// TIA Portal project "Bachelorarbeit Adrian Gehrig" (V15.1)
// Umsetzung des Smith Prädictor

(* hardware
DEVICE "S71500/ET200MP-Station_1"  S7-1500 station
   slot 0: "Profilschiene_0"  Rack  6ES7 590-1***0-0AA0
   slot 0: "PS 25W 24VDC_1"  PS 25W 24VDC  6ES7 505-0KA00-0AB0  V1.0
   slot 1: "PLC_1"  CPU 1515-2 PN  6ES7 515-2AM01-0AB0  V2.6
      slot 3: "CPU-Display_1"  6ES7591-1BA00-0AA0
*)

// ===== PLC "PLC_1"  CPU 1515-2 PN =====

TYPE "c_c_recursiveEstimat"
// *
//  * File: Smith_Predictor_MIAC.scl
//  *
//  * IEC 61131-3 Structured Text (ST) code generated for subsystem "Smith_Predictor_MIAC/Smith_Predictor_MIAC"
//  *
//  * Model name                      : Smith_Predictor_MIAC
//  * Model version                   : 1.3
//  * Model creator                   : Trips
//  * Model last modified by          : Trips
//  * Model last modified on          : Wed Mar 06 13:07:35 2019
//  * Model sample time               : 0s
//  * Subsystem name                  : Smith_Predictor_MIAC/Smith_Predictor_MIAC
//  * Subsystem sample time           : 1s
//  * Simulink PLC Coder version      : 2.6 (R2018b) 24-May-2018
//  * ST code generated on            : Wed Mar 06 13:15:01 2019
//  *
//  * Target IDE selection            : Siemens SIMATIC Step 7
//  * Test Bench included             : No
//  *
   STRUCT
      IteratorPosition : DInt;
   END_STRUCT;
END_TYPE

TYPE "c_d_recursiveEstimat"
   STRUCT
      OutputDataIterator : "c_c_recursiveEstimat";
      InputDataIterator : "c_c_recursiveEstimat";
   END_STRUCT;
END_TYPE

DATA_BLOCK "PT1_DB"   // DB1
{ S7_Optimized_Access := 'TRUE' }
VERSION : 0.1
// stored: InstanceOfName PT1
"PT1"
BEGIN
END_DATA_BLOCK

DATA_BLOCK "Signale"   // DB2
{ S7_Optimized_Access := 'TRUE' }
VERSION : 0.1
   VAR
      Input_PT1 : Real;
      Input_FOPDT : Real;
      Output_PT1 : Real;
      Output_FOPDT : Real;
      ssMethodType : Int;
      setpoint : Real;
      Start_Adaptation : Real;
      Hand_Value : Real;
      Enable_Auto : Real;
      Start_Identification : Real;
      Gain_Filtered : Real;
      Gain_Not_Filtered : Real;
      pulse_Indicatior : Bool;
      P_Controller : Real;
      I_Controller : Real;
   END_VAR
BEGIN
END_DATA_BLOCK

DATA_BLOCK "FOPDT_DB"   // DB3
{ S7_Optimized_Access := 'TRUE' }
VERSION : 0.1
// stored: InstanceOfName FOPDT
"FOPDT"
BEGIN
END_DATA_BLOCK

DATA_BLOCK "c_Smith_Predictor_MI_DB"   // DB4
{ S7_Optimized_Access := 'TRUE' }
VERSION : 0.1
// stored: InstanceOfName c_Smith_Predictor_MI
"c_Smith_Predictor_MI"
BEGIN
END_DATA_BLOCK

DATA_BLOCK "FOPDT_Tustin0_DB"   // DB5
{ S7_Optimized_Access := 'TRUE' }
VERSION : 0.1
// stored: InstanceOfName FOPDT_Tustin0
"FOPDT_Tustin0"
BEGIN
END_DATA_BLOCK

FUNCTION_BLOCK "PT1"   // FB1, SCL
{ S7_Optimized_Access := 'TRUE' }
VERSION : 0.1
// *
//  * File: TestPLCCoder.scl
//  *
//  * IEC 61131-3 Structured Text (ST) code generated for subsystem "TestPLCCoder/PT1"
//  *
//  * Model name                      : TestPLCCoder
//  * Model version                   : 1.1
//  * Model creator                   : Trips
//  * Model last modified by          : Trips
//  * Model last modified on          : Mon Feb 04 14:14:27 2019
//  * Model sample time               : 0.1s
//  * Subsystem name                  : TestPLCCoder/PT1
//  * Subsystem sample time           : 0.1s
//  * Simulink PLC Coder version      : 2.6 (R2018b) 24-May-2018
//  * ST code generated on            : Wed Feb 06 16:13:48 2019
//  *
//  * Target IDE selection            : Siemens SIMATIC Step 7
//  * Test Bench included             : No
//  *
   VAR_INPUT
      ssMethodType : Int;
      In1 : Real;
   END_VAR
   VAR_OUTPUT
      Out1 : Real;
   END_VAR
   VAR
      c_DiscreteTransferFc : Real;
   END_VAR
BEGIN
   CASE #ssMethodType OF
       0:
           (* InitializeConditions for DiscreteTransferFcn: '<S1>/Discrete Transfer Fcn1' *)
           #c_DiscreteTransferFc := 0.0;
       1:
           (* Outport: '<Root>/Out1' incorporates:
            *  DiscreteTransferFcn: '<S1>/Discrete Transfer Fcn1' *)
           #Out1 := 0.1 * #c_DiscreteTransferFc;
           (* Update for DiscreteTransferFcn: '<S1>/Discrete Transfer Fcn1' *)
           #c_DiscreteTransferFc := #In1 - (-0.9 * #c_DiscreteTransferFc);
   END_CASE;
END_FUNCTION_BLOCK

FUNCTION_BLOCK "FOPDT"   // FB2, SCL
{ S7_Optimized_Access := 'TRUE' }
VERSION : 0.1
// *
//  * File: FOPDT.scl
//  *
//  * IEC 61131-3 Structured Text (ST) code generated for subsystem "FOPDT/Subsystem"
//  *
//  * Model name                      : FOPDT
//  * Model version                   : 1.2
//  * Model creator                   : Trips
//  * Model last modified by          : Trips
//  * Model last modified on          : Tue Feb 26 09:05:07 2019
//  * Model sample time               : 1s
//  * Subsystem name                  : FOPDT/Subsystem
//  * Subsystem sample time           : 1s
//  * Simulink PLC Coder version      : 2.6 (R2018b) 24-May-2018
//  * ST code generated on            : Tue Feb 26 09:08:10 2019
//  *
//  * Target IDE selection            : Siemens SIMATIC Step 7
//  * Test Bench included             : No
//  *
   VAR_INPUT
      ssMethodType : Int;
      FOPD_Input : Real;
      Gain_System1 : Real;
      c_Time_Constant_Syst : Real;
      Sample_Time : Real;
      Dead_Time : DInt;
   END_VAR
   VAR_OUTPUT
      FOPD_Output : Real;
   END_VAR
   VAR
      Divide : Real;
      DiscreteTransferFcnv : Real;
      c_TmpSignalConversio : Array[0..1] of Real;
      Delay_DSTATE : Array[0..799] of Real;
      c_rtb_DiscreteTransf : Real;
      b_i : DInt;
   END_VAR
BEGIN
   CASE #ssMethodType OF
       0:
           (* InitializeConditions for DiscreteTransferFcn: '<S1>/Discrete Transfer Fcn' *)
           #DiscreteTransferFcnv := 0.0;
           (* InitializeConditions for Delay: '<S1>/Delay' *)
           FOR #b_i := 0 TO 799 DO
               #Delay_DSTATE[#b_i] := 0.0;
           END_FOR;
           (* End of InitializeConditions for Delay: '<S1>/Delay' *)
       1:
           (* Product: '<S1>/Divide' *)
           #Divide := #Gain_System1 / #c_Time_Constant_Syst;
           (* SignalConversion: '<S1>/TmpSignal ConversionAtDiscrete Transfer FcnInport3' incorporates:
            *  Constant: '<S1>/Constant'
            *  Gain: '<S1>/Gain'
            *  Gain: '<S1>/Gain1'
            *  Math: '<S1>/Exp'
            *  Product: '<S1>/Divide1'
            *
            * About '<S1>/Exp':
            *  Operator: exp *)
           #c_TmpSignalConversio[0] := 1.0;
           #c_TmpSignalConversio[1] := - EXP((- #Sample_Time) / #c_Time_Constant_Syst);
           (* DiscreteTransferFcn: '<S1>/Discrete Transfer Fcn' *)
           #c_rtb_DiscreteTransf := #Divide * #DiscreteTransferFcnv;
           (* Delay: '<S1>/Delay' *)
           IF #Dead_Time <= 0 THEN
               (* Outport: '<Root>/FOPD_Output' *)
               #FOPD_Output := #c_rtb_DiscreteTransf;
           ELSE
               IF #Dead_Time > 800 THEN
                   #b_i := 800;
               ELSE
                   #b_i := #Dead_Time;
               END_IF;
               (* Outport: '<Root>/FOPD_Output' *)
               #FOPD_Output := #Delay_DSTATE[800 - #b_i];
           END_IF;
           (* End of Delay: '<S1>/Delay' *)

           (* Update for DiscreteTransferFcn: '<S1>/Discrete Transfer Fcn' *)
           #DiscreteTransferFcnv := #FOPD_Input - (#c_TmpSignalConversio[1] * #DiscreteTransferFcnv);
           (* Update for Delay: '<S1>/Delay' *)
           FOR #b_i := 0 TO 798 DO
               #Delay_DSTATE[#b_i] := #Delay_DSTATE[#b_i + 1];
           END_FOR;
           #Delay_DSTATE[799] := #c_rtb_DiscreteTransf;
           (* End of Update for Delay: '<S1>/Delay' *)
   END_CASE;
END_FUNCTION_BLOCK

FUNCTION_BLOCK "ZCFCN_d_RISING"   // FB3, SCL
{ S7_Optimized_Access := 'TRUE' }
VERSION : 0.1
   VAR_INPUT
      u0 : Int;
      u1 : Real;
   END_VAR
   VAR_OUTPUT
      y0 : DInt;
      y1 : Int;
   END_VAR
   VAR
      rising : Bool;
      temp1 : Bool;
      temp2 : Bool;
   END_VAR
BEGIN
   #temp1 := FALSE;
   IF #u1 > 0.0 THEN
       #y1 := 1;
   ELSIF #u1 < 0.0 THEN
       #y1 := 2;
   ELSE
       #y1 := 0;
   END_IF;
   #temp2 := FALSE;
   IF #u0 = 2 THEN
       IF #y1 = 0 THEN
           #rising := TRUE;
       ELSIF #y1 = 1 THEN
           #rising := TRUE;
       ELSE
           #temp2 := TRUE;
       END_IF;
   ELSE
       #temp2 := TRUE;
   END_IF;
   IF #temp2 THEN
       IF #u0 = 0 THEN
           IF #y1 = 1 THEN
               #rising := TRUE;
           ELSE
               #temp1 := TRUE;
           END_IF;
       ELSE
           #temp1 := TRUE;
       END_IF;
   END_IF;
   IF #temp1 THEN
       IF #u0 = 101 THEN
           IF #y1 = 1 THEN
               #rising := TRUE;
           ELSE
               #rising := FALSE;
           END_IF;
       ELSE
           #rising := FALSE;
       END_IF;
   END_IF;
   IF #rising THEN
       #y0 := 1;
   ELSE
       #y0 := 0;
   END_IF;
   IF (#u0 = 2) AND (#y1 = 0) THEN
       #y1 := 100;
   END_IF;
END_FUNCTION_BLOCK

FUNCTION_BLOCK "Smith_Predictor_andv"   // FB4, SCL
{ S7_Optimized_Access := 'TRUE' }
VERSION : 0.1
   VAR_INPUT
      ssMethodType : Int;
      setpoint : Real;
      Dead_Time : Real;
      Y_Process : Real;
      Start_Adaption : Real;
      Hand_Value : Real;
      P_Controller : Real;
      I_Controller : Real;
      Gain_System : Real;
      Time_Constant_System : Real;
      Sample_Time : Real;
      Enable_Auto : Real;
      Start_Identification : Real;
   END_VAR
   VAR_OUTPUT
      Gain_Filtered : Real;
      Gain_Not_Filtered : Real;
      Controller_Output : Real;
   END_VAR
   VAR
      UnitDelay_DSTATE : Real;
      c_Numerator_ZTransfo : Real;
      c_Integrator_IC_LOAD : Int;
      Integrator_DSTATE : Real;
      c_Integrator_PrevRes : Int;
      c_inputSignalLowPass : Real;
      d_outputSignalLowPas : Real;
      icLoad : Int;
      icLoad_o : Int;
      icLoad_g : Int;
      icLoad_m : Int;
      icLoad_k : Int;
      icLoad_f : Int;
      c_EstimatedGainTiefp : Real;
      In1_i : Real;
      In1 : Real;
      In1_m : Real;
      c_System_Simulaton_s : Real;
      In1_b : Real;
      c_arxEstimator_not_e : Bool;
      arxEstimator : "c_d_recursiveEstimat";
      d_inputSignalLowPass : Int := 3;
      e_outputSignalLowPas : Int := 3;
      delayTheta_Reset_ZCE : Int := 3;
      delayL_Reset_ZCE : Int := 3;
      delayPhi_Reset_ZCE : Int := 3;
      c_delayBufferU_Reset : Int := 3;
      c_delayBufferY_Reset : Int := 3;
      c_delayBufferRegress : Int := 3;
      Delay_Reset_ZCE : Int := 3;
      d_EstimatedGainTiefp : Int := 3;
      c_System_Delay_Simul : Int := 3;
      c_System_Simulaton_R : Int := 3;
      d_System_Delay_Simul : Int := 3;
      e_System_Delay_Simul : Array[0..799] of Real;
      f_System_Delay_Simul : Array[0..799] of Real;
      c_Denumerator_ZTrans : Array[0..1] of Real;
      delayL_DSTATE : Array[0..8] of Real;
      delayTheta_DSTATE : Array[0..2] of Real;
      delayPhi_DSTATE : Array[0..3] of Real;
      c_InitialCovariancev : Array[0..8] of Real;
      i0_ZCFCN_d_RISING : "ZCFCN_d_RISING";
      phi : Array[0..2] of Real;
      fTr : Array[0..2] of Real;
      a1 : Real;
      sqrtA0overA1 : Real;
      sqrtA0timesA1 : Real;
      b_kk : DInt;
      rtb_UnitDelay : Real;
      rtb_theta : Array[0..2] of Real;
      rtb_L : Array[0..8] of Real;
      rtb_phiMemory : Array[0..3] of Real;
      imputdelayedminus : Real;
      input : Real;
      c_outputSignalLowPas : Real;
      rtb_theta_tmp : Real;
      rtb_theta_tmp_0 : Real;
   END_VAR
   // c_InitialCovariancev[0] := 3.162278;
   // c_InitialCovariancev[1] := 0.0;
   // c_InitialCovariancev[2] := 0.0;
   // c_InitialCovariancev[3] := 0.0;
   // c_InitialCovariancev[4] := 3.162278;
   // c_InitialCovariancev[5] := 0.0;
   // c_InitialCovariancev[6] := 0.0;
   // c_InitialCovariancev[7] := 0.0;
   // c_InitialCovariancev[8] := 3.162278;
BEGIN
   CASE #ssMethodType OF
       0:
           (* InitializeConditions for UnitDelay: '<S1>/Unit Delay' *)
           #UnitDelay_DSTATE := 0.0;
           (* SystemInitialize for Atomic SubSystem: '<S1>/System Identification' *)
           (* InitializeConditions for DiscreteTransferFcn: '<S3>/input Signal Low Pass Filter' *)
           #c_inputSignalLowPass := 0.0;
           (* InitializeConditions for DiscreteTransferFcn: '<S3>/output Signal Low Pass Filter1' *)
           #d_outputSignalLowPas := 0.0;
           (* InitializeConditions for Delay: '<S106>/delayTheta' *)
           #icLoad := 1;
           (* InitializeConditions for Delay: '<S106>/delayL' *)
           #icLoad_o := 1;
           (* InitializeConditions for Delay: '<S106>/delayPhi' *)
           #icLoad_g := 1;
           (* InitializeConditions for Delay: '<S106>/delayBufferU' *)
           #icLoad_m := 1;
           (* InitializeConditions for Delay: '<S106>/delayBufferY' *)
           #icLoad_k := 1;
           (* InitializeConditions for Delay: '<S126>/delayBufferRegressors' *)
           #icLoad_f := 1;
           (* InitializeConditions for DiscreteTransferFcn: '<S3>/Estimated Gain Tiefpassfilter' *)
           #c_EstimatedGainTiefp := 0.0;
           (* SystemInitialize for MATLAB Function: '<S126>/rarx' *)
           #c_arxEstimator_not_e := FALSE;
           (* SystemInitialize for Enabled SubSystem: '<S3>/Get_Current_Output_Offset' *)
           (* SystemInitialize for Outport: '<S104>/Hold when disabled' *)
           #In1_i := 0.0;
           (* End of SystemInitialize for SubSystem: '<S3>/Get_Current_Output_Offset' *)

           (* SystemInitialize for Enabled SubSystem: '<S3>/Get_Current_delayed_Input_Offset' *)
           (* SystemInitialize for Outport: '<S105>/Hold when disabled' *)
           #In1 := 0.0;
           (* End of SystemInitialize for SubSystem: '<S3>/Get_Current_delayed_Input_Offset' *)
           (* End of SystemInitialize for SubSystem: '<S1>/System Identification' *)

           (* SystemInitialize for Atomic SubSystem: '<S1>/Adaptive SmithPredictor1' *)
           (* InitializeConditions for DiscreteTransferFcn: '<S2>/System_Simulaton' *)
           #c_System_Simulaton_s := 0.0;
           (* End of SystemInitialize for SubSystem: '<S1>/Adaptive SmithPredictor1' *)
           (* SystemInitialize for Atomic SubSystem: '<S1>/Adaptive SmithPredictor1' *)
           (* SystemInitialize for Atomic SubSystem: '<S1>/System Identification' *)
           FOR #b_kk := 0 TO 799 DO
               (* InitializeConditions for Delay: '<S3>/System_Delay_Simulation' *)
               #e_System_Delay_Simul[#b_kk] := 0.0;
               (* InitializeConditions for Delay: '<S2>/System_Delay_Simulation' *)
               #f_System_Delay_Simul[#b_kk] := 0.0;
           END_FOR;
           (* End of SystemInitialize for SubSystem: '<S1>/System Identification' *)

           (* InitializeConditions for DiscreteIntegrator: '<S61>/Integrator' *)
           #c_Integrator_IC_LOAD := 1;
           #c_Integrator_PrevRes := 2;
           (* SystemInitialize for Enabled SubSystem: '<S2>/Get_Current_Offset1' *)
           (* SystemInitialize for Outport: '<S5>/Hold when disabled' *)
           #In1_m := 0.0;
           (* End of SystemInitialize for SubSystem: '<S2>/Get_Current_Offset1' *)

           (* SystemInitialize for Enabled SubSystem: '<S2>/Get_Current_Offset' *)
           (* SystemInitialize for Outport: '<S4>/Hold when disabled' *)
           #In1_b := 0.0;
           (* End of SystemInitialize for SubSystem: '<S2>/Get_Current_Offset' *)
           (* End of SystemInitialize for SubSystem: '<S1>/Adaptive SmithPredictor1' *)
       1:
           (* UnitDelay: '<S1>/Unit Delay' *)
           #rtb_UnitDelay := #UnitDelay_DSTATE;
           (* Outputs for Atomic SubSystem: '<S1>/System Identification' *)
           (* DiscreteTransferFcn: '<S3>/input Signal Low Pass Filter' *)
           #i0_ZCFCN_d_RISING(u0 := #d_inputSignalLowPass,
                              u1 := #Start_Identification);
           #b_kk := #i0_ZCFCN_d_RISING.y0;
           #d_inputSignalLowPass := #i0_ZCFCN_d_RISING.y1;
           IF #b_kk <> 0 THEN
               #c_inputSignalLowPass := 0.0;
           END_IF;
           #input := 0.01 * #c_inputSignalLowPass;
           (* End of DiscreteTransferFcn: '<S3>/input Signal Low Pass Filter' *)

           (* DiscreteTransferFcn: '<S3>/output Signal Low Pass Filter1' *)
           #i0_ZCFCN_d_RISING(u0 := #e_outputSignalLowPas,
                              u1 := #Start_Identification);
           #b_kk := #i0_ZCFCN_d_RISING.y0;
           #e_outputSignalLowPas := #i0_ZCFCN_d_RISING.y1;
           IF #b_kk <> 0 THEN
               #d_outputSignalLowPas := 0.0;
           END_IF;
           #imputdelayedminus := 0.01 * #d_outputSignalLowPas;
           #c_outputSignalLowPas := #imputdelayedminus;
           (* Delay: '<S106>/delayTheta' *)
           #i0_ZCFCN_d_RISING(u0 := #delayTheta_Reset_ZCE,
                              u1 := #Start_Identification);
           #b_kk := #i0_ZCFCN_d_RISING.y0;
           #delayTheta_Reset_ZCE := #i0_ZCFCN_d_RISING.y1;
           IF #b_kk <> 0 THEN
               #icLoad := 1;
           END_IF;
           IF #icLoad <> 0 THEN
               #delayTheta_DSTATE[0] := 2.2204460492503131E-16;
               #delayTheta_DSTATE[1] := 2.2204460492503131E-16;
               #delayTheta_DSTATE[2] := 2.2204460492503131E-16;
           END_IF;
           (* Delay: '<S106>/delayL' incorporates:
            *  Constant: '<S106>/InitialCovariance' *)
           #i0_ZCFCN_d_RISING(u0 := #delayL_Reset_ZCE,
                              u1 := #Start_Identification);
           #b_kk := #i0_ZCFCN_d_RISING.y0;
           #delayL_Reset_ZCE := #i0_ZCFCN_d_RISING.y1;
           IF #b_kk <> 0 THEN
               #icLoad_o := 1;
           END_IF;
           IF #icLoad_o <> 0 THEN
               FOR #b_kk := 0 TO 8 DO
                   #delayL_DSTATE[#b_kk] := #c_InitialCovariancev[#b_kk];
               END_FOR;
           END_IF;
           (* Delay: '<S106>/delayPhi' *)
           #i0_ZCFCN_d_RISING(u0 := #delayPhi_Reset_ZCE,
                              u1 := #Start_Identification);
           #b_kk := #i0_ZCFCN_d_RISING.y0;
           #delayPhi_Reset_ZCE := #i0_ZCFCN_d_RISING.y1;
           IF #b_kk <> 0 THEN
               #icLoad_g := 1;
           END_IF;
           IF #icLoad_g <> 0 THEN
               #delayPhi_DSTATE[0] := 0.0;
               #delayPhi_DSTATE[1] := 0.0;
               #delayPhi_DSTATE[2] := 0.0;
               #delayPhi_DSTATE[3] := 0.0;
           END_IF;
           (* Delay: '<S106>/delayBufferU' *)
           #i0_ZCFCN_d_RISING(u0 := #c_delayBufferU_Reset,
                              u1 := #Start_Identification);
           #b_kk := #i0_ZCFCN_d_RISING.y0;
           #c_delayBufferU_Reset := #i0_ZCFCN_d_RISING.y1;
           IF #b_kk <> 0 THEN
               #icLoad_m := 1;
           END_IF;
           (* End of Delay: '<S106>/delayBufferU' *)

           (* Delay: '<S106>/delayBufferY' *)
           #i0_ZCFCN_d_RISING(u0 := #c_delayBufferY_Reset,
                              u1 := #Start_Identification);
           #b_kk := #i0_ZCFCN_d_RISING.y0;
           #c_delayBufferY_Reset := #i0_ZCFCN_d_RISING.y1;
           IF #b_kk <> 0 THEN
               #icLoad_k := 1;
           END_IF;
           (* End of Delay: '<S106>/delayBufferY' *)

           (* Delay: '<S126>/delayBufferRegressors' *)
           #i0_ZCFCN_d_RISING(u0 := #c_delayBufferRegress,
                              u1 := #Start_Identification);
           #b_kk := #i0_ZCFCN_d_RISING.y0;
           #c_delayBufferRegress := #i0_ZCFCN_d_RISING.y1;
           IF #b_kk <> 0 THEN
               #icLoad_f := 1;
           END_IF;
           (* End of Delay: '<S126>/delayBufferRegressors' *)

           (* Delay: '<S128>/Delay' *)
           #i0_ZCFCN_d_RISING(u0 := #Delay_Reset_ZCE,
                              u1 := #Start_Identification);
           #b_kk := #i0_ZCFCN_d_RISING.y0;
           #Delay_Reset_ZCE := #i0_ZCFCN_d_RISING.y1;
           (* MATLAB Function: '<S126>/rarx' *)
           (* % Was a reset trigered? *)
           (* MATLAB Function 'Recursive Estimation/rarx/rarx': '<S135>:1' *)
           (* Copyright 2015-2018 The MathWorks, Inc. *)
           (* Get the estimator object. Use the arx estimator with nb=0 *)
           (* '<S135>:1:17' if isempty(arxEstimator) *)
           IF NOT #c_arxEstimator_not_e THEN
               (* '<S135>:1:18' arxEstimator = recursiveEstimation.internal.rpoly.getEstimator(... *)
               (* '<S135>:1:19'         'arx',... *)
               (* '<S135>:1:20'         algorithmParams); *)
               #c_arxEstimator_not_e := TRUE;
           END_IF;
           (* If user triggered a reset, communicate this to the estimator *)
           (* '<S135>:1:24' if hasTriggeredReset *)
           (* Update algorithm states, perform estimation *)
           (* % States *)
           (* % new IO data *)
           (* '<S135>:1:31' [phiMemory, uMemory, yMemory, regressorsMemory, ... *)
           (* '<S135>:1:32'     theta, L, ... *)
           (* '<S135>:1:33'     A, B, e] = ... *)
           (* '<S135>:1:34'     arxEstimator.estimate(... *)
           (* '<S135>:1:35'     phiMemory, uMemory, yMemory, regressorsMemory, theta, L, ... % States *)
           (* '<S135>:1:36'     yMeas, uMeas,... % new IO data *)
           (* '<S135>:1:37'     isEnabled, adg1, adg2, algorithmParams); *)
           #arxEstimator.OutputDataIterator.IteratorPosition := 1;
           #arxEstimator.InputDataIterator.IteratorPosition := 1;
           #arxEstimator.OutputDataIterator.IteratorPosition := MIN(IN1 := #arxEstimator.OutputDataIterator.IteratorPosition + 1,
                                                                    IN2 := 2);
           #arxEstimator.InputDataIterator.IteratorPosition := MIN(IN1 := #arxEstimator.InputDataIterator.IteratorPosition + 1,
                                                                   IN2 := 2);
           (* End of Outputs for SubSystem: '<S1>/System Identification' *)
           (* Outputs for Atomic SubSystem: '<S1>/System Identification' *)
           (* MATLAB Function: '<S126>/rarx' incorporates:
            *  DataTypeConversion: '<S106>/DataTypeConversionEnable'
            *  Delay: '<S106>/delayL'
            *  Delay: '<S106>/delayPhi'
            *  Delay: '<S106>/delayTheta'
            *  DiscreteTransferFcn: '<S3>/output Signal Low Pass Filter1' *)
           FOR #b_kk := 0 TO 8 DO
               #rtb_L[#b_kk] := #delayL_DSTATE[#b_kk];
           END_FOR;
           #rtb_theta[0] := #delayTheta_DSTATE[0];
           #rtb_theta[1] := #delayTheta_DSTATE[1];
           #rtb_theta[2] := #delayTheta_DSTATE[2];
           #imputdelayedminus := #imputdelayedminus - (((#delayPhi_DSTATE[0] * #delayTheta_DSTATE[0]) + (#delayPhi_DSTATE[1] * #delayTheta_DSTATE[1])
           ) + (#delayPhi_DSTATE[3] * #delayTheta_DSTATE[2]));
           IF #Start_Identification <> 0.0 THEN
               FOR #b_kk := 0 TO 2 DO
                   #fTr[#b_kk] := (#delayL_DSTATE[(3 * #b_kk) + 2] * #delayPhi_DSTATE[3]) + ((#delayL_DSTATE[(3 * #b_kk) + 1] * #delayPhi_DSTATE[1])
                   + (#delayL_DSTATE[3 * #b_kk] * #delayPhi_DSTATE[0]));
               END_FOR;
               #phi[0] := 0.0;
               #rtb_theta[0] := 0.0;
               #phi[1] := 0.0;
               #rtb_theta[1] := 0.0;
               #a1 := (#fTr[2] * #fTr[2]) + 1.0;
               #sqrtA0overA1 := SQRT(1.0 / #a1);
               #rtb_theta[2] := #rtb_L[8] * #fTr[2];
               #rtb_L[8] := (#rtb_L[8] * #sqrtA0overA1) - (0.0 / (#sqrtA0overA1 * #a1));
               #phi[2] := #rtb_theta[2];
               #sqrtA0overA1 := #a1;
               #a1 := (#fTr[1] * #fTr[1]) + #a1;
               #sqrtA0overA1 := SQRT(#sqrtA0overA1 / #a1);
               #sqrtA0timesA1 := #sqrtA0overA1 * #a1;
               FOR #b_kk := 0 TO 1 DO
                   #rtb_theta_tmp := #rtb_L[5 - #b_kk];
                   #rtb_theta_tmp_0 := #phi[2 - #b_kk];
                   #rtb_theta[2 - #b_kk] := (#rtb_theta_tmp * #fTr[1]) + #rtb_theta_tmp_0;
                   #rtb_L[5 - #b_kk] := (#rtb_theta_tmp * #sqrtA0overA1) - ((#rtb_theta_tmp_0 * #fTr[1]) / #sqrtA0timesA1);
                   #phi[2 - #b_kk] := #rtb_theta[2 - #b_kk];
               END_FOR;
               #sqrtA0overA1 := #a1;
               #a1 := (#fTr[0] * #fTr[0]) + #a1;
               #sqrtA0overA1 := SQRT(#sqrtA0overA1 / #a1);
               #sqrtA0timesA1 := #sqrtA0overA1 * #a1;
               FOR #b_kk := 0 TO 2 DO
                   #rtb_theta_tmp := #rtb_L[2 - #b_kk];
                   #rtb_theta_tmp_0 := #phi[2 - #b_kk];
                   #rtb_theta[2 - #b_kk] := (#rtb_theta_tmp * #fTr[0]) + #rtb_theta_tmp_0;
                   #rtb_L[2 - #b_kk] := (#rtb_theta_tmp * #sqrtA0overA1) - ((#rtb_theta_tmp_0 * #fTr[0]) / #sqrtA0timesA1);
                   #phi[2 - #b_kk] := #rtb_theta[2 - #b_kk];
               END_FOR;
               #rtb_theta[0] := #rtb_theta[0] / #a1;
               #rtb_theta[1] := #rtb_theta[1] / #a1;
               #rtb_theta[0] := (#rtb_theta[0] * #imputdelayedminus) + #delayTheta_DSTATE[0];
               #rtb_theta[1] := (#rtb_theta[1] * #imputdelayedminus) + #delayTheta_DSTATE[1];
               #rtb_theta[2] := ((#rtb_theta[2] / #a1) * #imputdelayedminus) + #delayTheta_DSTATE[2];
           END_IF;
           #rtb_phiMemory[2] := #delayPhi_DSTATE[1];
           #rtb_phiMemory[1] := #delayPhi_DSTATE[0];
           (* Outputs for Atomic SubSystem: '<S3>/Calculate DC Gain1' *)
           (* Product: '<S103>/Divide' incorporates:
            *  MATLAB Function: '<S126>/rarx'
            *  Sum: '<S103>/A(z) Sum of Elements' *)
            (* helper variables *)
           #a1 := #rtb_theta[2] / ((1.0 + #rtb_theta[0]) + #rtb_theta[1]);
           (* Saturate: '<S103>/Gain_Saturation' incorporates:
            *  Outport: '<Root>/Gain_Filtered' *)
           IF #a1 >= 1.5 THEN
               #Gain_Filtered := 1.5;
           ELSIF #a1 > 0.01 THEN
               #Gain_Filtered := #a1;
           ELSE
               #Gain_Filtered := 0.01;
           END_IF;
           (* End of Saturate: '<S103>/Gain_Saturation' *)
           (* End of Outputs for SubSystem: '<S3>/Calculate DC Gain1' *)

           (* DiscreteTransferFcn: '<S3>/Estimated Gain Tiefpassfilter' incorporates:
            *  Constant: '<S3>/Constant3' *)
           #i0_ZCFCN_d_RISING(u0 := #d_EstimatedGainTiefp,
                              u1 := #Start_Identification);
           #b_kk := #i0_ZCFCN_d_RISING.y0;
           #d_EstimatedGainTiefp := #i0_ZCFCN_d_RISING.y1;
           IF #b_kk <> 0 THEN
               #c_EstimatedGainTiefp := 0.0;
           END_IF;
           #sqrtA0overA1 := 0.00083333333333333339 * #c_EstimatedGainTiefp;
           (* End of DiscreteTransferFcn: '<S3>/Estimated Gain Tiefpassfilter' *)

           (* Outputs for Enabled SubSystem: '<S3>/Get_Current_Output_Offset' incorporates:
            *  EnablePort: '<S104>/Enable' *)
            (* Logic: '<S3>/NOT' incorporates:
             *  Inport: '<S104>/In1' *)
           IF #Start_Identification = 0.0 THEN
               #In1_i := #Y_Process;
           END_IF;
           (* End of Logic: '<S3>/NOT' *)
           (* End of Outputs for SubSystem: '<S3>/Get_Current_Output_Offset' *)

           (* Delay: '<S3>/System_Delay_Simulation' incorporates:
            *  Constant: '<S3>/Vorsicht wenn resettet wird muss erst dieser Totzeitspeicher  voll gelaufen sein bevor die Adaption starten darf  Sonst kommt heir immer 0 raus und die Identifikation kann nicht rechnen' *)
           #i0_ZCFCN_d_RISING(u0 := #c_System_Delay_Simul,
                              u1 := 0.0);
           #b_kk := #i0_ZCFCN_d_RISING.y0;
           #c_System_Delay_Simul := #i0_ZCFCN_d_RISING.y1;
           IF #b_kk <> 0 THEN
               FOR #b_kk := 0 TO 799 DO
                   #e_System_Delay_Simul[#b_kk] := 0.0;
               END_FOR;
           END_IF;
           IF #Dead_Time < 1.0 THEN
               #a1 := #rtb_UnitDelay;
           ELSE
               IF #Dead_Time > 800.0 THEN
                   #b_kk := 800;
               ELSE
                   #b_kk := TRUNC(#Dead_Time);
               END_IF;
               #a1 := #e_System_Delay_Simul[800 - #b_kk];
           END_IF;
           (* End of Delay: '<S3>/System_Delay_Simulation' *)

           (* Outputs for Enabled SubSystem: '<S3>/Get_Current_delayed_Input_Offset' incorporates:
            *  EnablePort: '<S105>/Enable' *)
            (* Logic: '<S3>/NOT1' incorporates:
             *  Inport: '<S105>/In1' *)
           IF #Start_Identification = 0.0 THEN
               #In1 := #a1;
           END_IF;
           (* End of Logic: '<S3>/NOT1' *)
           (* End of Outputs for SubSystem: '<S3>/Get_Current_delayed_Input_Offset' *)

           (* Update for DiscreteTransferFcn: '<S3>/input Signal Low Pass Filter' incorporates:
            *  Sum: '<S3>/Substract Current Offset  so that the linearised model works1' *)
           #c_inputSignalLowPass := (#a1 - #In1) - (-0.99 * #c_inputSignalLowPass);
           (* Update for DiscreteTransferFcn: '<S3>/output Signal Low Pass Filter1' incorporates:
            *  Sum: '<S3>/Substract Current Offset  so that the linearised model works' *)
           #d_outputSignalLowPas := (#Y_Process - #In1_i) - (-0.99 * #d_outputSignalLowPas);
           (* Update for Delay: '<S106>/delayTheta' *)
           #icLoad := 0;
           #delayTheta_DSTATE[0] := #rtb_theta[0];
           #delayTheta_DSTATE[1] := #rtb_theta[1];
           #delayTheta_DSTATE[2] := #rtb_theta[2];
           (* Update for Delay: '<S106>/delayL' *)
           #icLoad_o := 0;
           (* End of Outputs for SubSystem: '<S1>/System Identification' *)
           (* Outputs for Atomic SubSystem: '<S1>/System Identification' *)
           (* Update for Delay: '<S106>/delayL' *)
           FOR #b_kk := 0 TO 8 DO
               #delayL_DSTATE[#b_kk] := #rtb_L[#b_kk];
           END_FOR;
           (* Update for Delay: '<S106>/delayPhi' incorporates:
            *  MATLAB Function: '<S126>/rarx' *)
           #icLoad_g := 0;
           #delayPhi_DSTATE[0] := - #c_outputSignalLowPas;
           #delayPhi_DSTATE[1] := #rtb_phiMemory[1];
           #delayPhi_DSTATE[2] := #rtb_phiMemory[2];
           #delayPhi_DSTATE[3] := #input;
           (* Update for Delay: '<S106>/delayBufferU' *)
           #icLoad_m := 0;
           (* Update for Delay: '<S106>/delayBufferY' *)
           #icLoad_k := 0;
           (* Update for Delay: '<S126>/delayBufferRegressors' *)
           #icLoad_f := 0;
           (* Update for DiscreteTransferFcn: '<S3>/Estimated Gain Tiefpassfilter' incorporates:
            *  Outport: '<Root>/Gain_Filtered' *)
           #c_EstimatedGainTiefp := #Gain_Filtered - (-0.99916701379245831 * #c_EstimatedGainTiefp);
           (* Update for Delay: '<S3>/System_Delay_Simulation' *)
           FOR #b_kk := 0 TO 798 DO
               #e_System_Delay_Simul[#b_kk] := #e_System_Delay_Simul[#b_kk + 1];
           END_FOR;
           #e_System_Delay_Simul[799] := #rtb_UnitDelay;
           (* End of Update for Delay: '<S3>/System_Delay_Simulation' *)
           (* End of Outputs for SubSystem: '<S1>/System Identification' *)

           (* Outport: '<Root>/Gain_Not_Filtered' *)
           #Gain_Not_Filtered := #sqrtA0overA1;
           (* Outputs for Atomic SubSystem: '<S1>/Adaptive SmithPredictor1' *)
           (* Product: '<S2>/Divide' incorporates:
            *  Constant: '<S2>/Constant1' *)
           #c_Numerator_ZTransfo := 1.0 / #Time_Constant_System;
           (* Switch: '<S2>/Hand_Mode2' incorporates:
            *  Constant: '<S2>/Constant2' *)
           IF #Enable_Auto > 0.0 THEN
               #a1 := #setpoint;
           ELSE
               #a1 := 0.0;
           END_IF;
           (* End of Switch: '<S2>/Hand_Mode2' *)

           (* Outputs for Enabled SubSystem: '<S2>/Get_Current_Offset1' incorporates:
            *  EnablePort: '<S5>/Enable' *)
            (* Logic: '<S2>/NOT1' incorporates:
             *  Inport: '<S5>/In1' *)
           IF #Enable_Auto = 0.0 THEN
               #In1_m := #Y_Process;
           END_IF;
           (* End of Logic: '<S2>/NOT1' *)
           (* End of Outputs for SubSystem: '<S2>/Get_Current_Offset1' *)

           (* Switch: '<S2>/Hand_Mode4' incorporates:
            *  Constant: '<S2>/Constant5' *)
           IF #Enable_Auto > 0.0 THEN
               #rtb_UnitDelay := #In1_m;
           ELSE
               #rtb_UnitDelay := 0.0;
           END_IF;
           (* End of Switch: '<S2>/Hand_Mode4' *)

           (* Sum: '<S2>/Substract Current Setpoint Offset' *)
           #c_outputSignalLowPas := #a1 - #rtb_UnitDelay;
           (* SignalConversion: '<S2>/TmpSignal ConversionAtSystem_SimulatonInport3' incorporates:
            *  Constant: '<S2>/Constant'
            *  Gain: '<S2>/Gain'
            *  Gain: '<S2>/Gain1'
            *  Math: '<S2>/Exp'
            *  Product: '<S2>/Divide1'
            *
            * About '<S2>/Exp':
            *  Operator: exp *)
           #c_Denumerator_ZTrans[0] := 1.0;
           #c_Denumerator_ZTrans[1] := - EXP((- #Sample_Time) / #Time_Constant_System);
           (* DiscreteTransferFcn: '<S2>/System_Simulaton' *)
           #i0_ZCFCN_d_RISING(u0 := #c_System_Simulaton_R,
                              u1 := #Enable_Auto);
           #b_kk := #i0_ZCFCN_d_RISING.y0;
           #c_System_Simulaton_R := #i0_ZCFCN_d_RISING.y1;
           IF #b_kk <> 0 THEN
               #c_System_Simulaton_s := 0.0;
           END_IF;
           #input := #c_Numerator_ZTransfo * #c_System_Simulaton_s;
           (* End of DiscreteTransferFcn: '<S2>/System_Simulaton' *)

           (* Delay: '<S2>/System_Delay_Simulation' *)
           #i0_ZCFCN_d_RISING(u0 := #d_System_Delay_Simul,
                              u1 := #Enable_Auto);
           #b_kk := #i0_ZCFCN_d_RISING.y0;
           #d_System_Delay_Simul := #i0_ZCFCN_d_RISING.y1;
           IF #b_kk <> 0 THEN
               FOR #b_kk := 0 TO 799 DO
                   #f_System_Delay_Simul[#b_kk] := 0.0;
               END_FOR;
           END_IF;
           IF #Dead_Time < 1.0 THEN
               #imputdelayedminus := #input;
           ELSE
               IF #Dead_Time > 800.0 THEN
                   #b_kk := 800;
               ELSE
                   #b_kk := TRUNC(#Dead_Time);
               END_IF;
               #imputdelayedminus := #f_System_Delay_Simul[800 - #b_kk];
           END_IF;
           (* End of Delay: '<S2>/System_Delay_Simulation' *)

           (* Switch: '<S2>/Hand_Mode3' incorporates:
            *  Constant: '<S2>/Constant3' *)
           IF #Enable_Auto > 0.0 THEN
               #a1 := #Y_Process;
           ELSE
               #a1 := 0.0;
           END_IF;
           (* End of Switch: '<S2>/Hand_Mode3' *)

           (* Sum: '<S2>/Sum' incorporates:
            *  Sum: '<S2>/Substract Current Offset  so that the linearised model works1'
            *  Sum: '<S2>/Sum17'
            *  Sum: '<S2>/Sum18' *)
           #rtb_UnitDelay := #c_outputSignalLowPas - (((#a1 - #rtb_UnitDelay) - #imputdelayedminus) + #input);
           (* DiscreteIntegrator: '<S61>/Integrator' *)
           IF #c_Integrator_IC_LOAD <> 0 THEN
               #Integrator_DSTATE := #Hand_Value;
           END_IF;
           IF (#Enable_Auto > 0.0) AND (#c_Integrator_PrevRes <= 0) THEN
               #Integrator_DSTATE := #Hand_Value;
           END_IF;
           (* Sum: '<S90>/Sum' incorporates:
            *  DiscreteIntegrator: '<S61>/Integrator'
            *  Product: '<S77>/PProd Out' *)
           #a1 := (#rtb_UnitDelay * #P_Controller) + #Integrator_DSTATE;
           (* Saturate: '<S82>/Saturation' *)
           IF #a1 >= 100.0 THEN
               #a1 := 100.0;
           ELSIF #a1 <= 0.0 THEN
               #a1 := 0.0;
           END_IF;
           (* End of Saturate: '<S82>/Saturation' *)

           (* Switch: '<S2>/Hand_Mode' *)
           IF #Enable_Auto > 0.0 THEN
               #Controller_Output := #a1;
           ELSE
               #Controller_Output := #Hand_Value;
           END_IF;
           (* End of Switch: '<S2>/Hand_Mode' *)

           (* Outputs for Enabled SubSystem: '<S2>/Get_Current_Offset' incorporates:
            *  EnablePort: '<S4>/Enable' *)
            (* Logic: '<S2>/NOT' incorporates:
             *  Inport: '<S4>/In1' *)
           IF #Enable_Auto = 0.0 THEN
               #In1_b := #Controller_Output;
           END_IF;
           (* End of Logic: '<S2>/NOT' *)
           (* End of Outputs for SubSystem: '<S2>/Get_Current_Offset' *)

           (* Switch: '<S2>/Hand_Mode1' incorporates:
            *  Constant: '<S2>/Constant4'
            *  Sum: '<S2>/Substract Current Offset  so that the linearised model works' *)
           IF #Enable_Auto > 0.0 THEN
               #a1 := #Controller_Output - #In1_b;
           ELSE
               #a1 := 0.0;
           END_IF;
           (* End of Switch: '<S2>/Hand_Mode1' *)

           (* Switch: '<S2>/Switch_from_initial_Gain_to_Estimated' *)
           IF #Start_Adaption <= 0.0 THEN
               #sqrtA0overA1 := #Gain_System;
           END_IF;
           (* End of Switch: '<S2>/Switch_from_initial_Gain_to_Estimated' *)

           (* Product: '<S2>/Mul_Gain_or_Estimate' *)
           #sqrtA0overA1 := #a1 * #sqrtA0overA1;
           (* Update for DiscreteTransferFcn: '<S2>/System_Simulaton' *)
           #c_System_Simulaton_s := #sqrtA0overA1 - (#c_Denumerator_ZTrans[1] * #c_System_Simulaton_s);
           (* Update for Delay: '<S2>/System_Delay_Simulation' *)
           FOR #b_kk := 0 TO 798 DO
               #f_System_Delay_Simul[#b_kk] := #f_System_Delay_Simul[#b_kk + 1];
           END_FOR;
           #f_System_Delay_Simul[799] := #input;
           (* End of Update for Delay: '<S2>/System_Delay_Simulation' *)

           (* Update for DiscreteIntegrator: '<S61>/Integrator' incorporates:
            *  Product: '<S50>/IProd Out' *)
           #c_Integrator_IC_LOAD := 0;
           #Integrator_DSTATE := (#rtb_UnitDelay * #I_Controller) + #Integrator_DSTATE;
           IF #Enable_Auto > 0.0 THEN
               #c_Integrator_PrevRes := 1;
           ELSIF #Enable_Auto < 0.0 THEN
               #c_Integrator_PrevRes := -1;
           ELSIF #Enable_Auto = 0.0 THEN
               #c_Integrator_PrevRes := 0;
           ELSE
               #c_Integrator_PrevRes := 2;
           END_IF;
           (* End of Update for DiscreteIntegrator: '<S61>/Integrator' *)
           (* End of Outputs for SubSystem: '<S1>/Adaptive SmithPredictor1' *)

           (* Update for UnitDelay: '<S1>/Unit Delay' *)
           #UnitDelay_DSTATE := #Controller_Output;
   END_CASE;
END_FUNCTION_BLOCK

FUNCTION_BLOCK "FOPDT_Tustin0"   // FB5, SCL
{ S7_Optimized_Access := 'TRUE' }
VERSION : 0.1
// *
//  * File: FOPDT_Tustin.scl
//  *
//  * IEC 61131-3 Structured Text (ST) code generated for subsystem "FOPDT_Tustin/FOPDT_Tustin"
//  *
//  * Model name                      : FOPDT_Tustin
//  * Model version                   : 1.11
//  * Model creator                   : Trips
//  * Model last modified by          : Trips
//  * Model last modified on          : Mon Mar 04 23:33:50 2019
//  * Model sample time               : 1s
//  * Subsystem name                  : FOPDT_Tustin/FOPDT_Tustin
//  * Subsystem sample time           : 1s
//  * Simulink PLC Coder version      : 2.6 (R2018b) 24-May-2018
//  * ST code generated on            : Mon Mar 04 23:34:12 2019
//  *
//  * Target IDE selection            : Siemens SIMATIC Step 7
//  * Test Bench included             : No
//  *
   VAR_INPUT
      ssMethodType : Int;
      FOPD_Input : Real;
      Gain_System : Real;
      Time_Constant_System : Real;
      Sample_Time : Real;
      Dead_Time : Real;
   END_VAR
   VAR_OUTPUT
      FOPD_Output : Real;
   END_VAR
   VAR
      DiscreteTransferFcnv : Real;
      c_TmpSignalConversio : Array[0..1] of Real;
      Delay_DSTATE : Array[0..799] of Real;
      d_TmpSignalConversio : Array[0..1] of Real;
      rtb_Gain : Real;
      rtb_Divide : Real;
      b_i : DInt;
   END_VAR
BEGIN
   CASE #ssMethodType OF
       0:
           (* InitializeConditions for DiscreteTransferFcn: '<S1>/Discrete Transfer Fcn' *)
           #DiscreteTransferFcnv := 0.0;
           (* InitializeConditions for Delay: '<S1>/Delay' *)
           FOR #b_i := 0 TO 799 DO
               #Delay_DSTATE[#b_i] := 0.0;
           END_FOR;
           (* End of InitializeConditions for Delay: '<S1>/Delay' *)
       1:
           (* Gain: '<S1>/Gain' *)
           #rtb_Gain := 2.0 * #Time_Constant_System;
           (* Product: '<S1>/Divide' incorporates:
            *  Product: '<S1>/Multiply'
            *  Sum: '<S1>/Add' *)
           #rtb_Divide := (#Gain_System * #Sample_Time) / (#Sample_Time + #rtb_Gain);
           (* SignalConversion: '<S1>/TmpSignal ConversionAtDiscrete Transfer FcnInport2' *)
           #c_TmpSignalConversio[0] := #rtb_Divide;
           #c_TmpSignalConversio[1] := #rtb_Divide;
           (* SignalConversion: '<S1>/TmpSignal ConversionAtDiscrete Transfer FcnInport3' incorporates:
            *  Constant: '<S1>/Constant'
            *  Gain: '<S1>/Gain1'
            *  Product: '<S1>/Divide1'
            *  Sum: '<S1>/Add1'
            *  Sum: '<S1>/Minus' *)
           #d_TmpSignalConversio[0] := 1.0;
           #d_TmpSignalConversio[1] := - ((#rtb_Gain - #Sample_Time) / (#rtb_Gain + #Sample_Time));
           (* DiscreteTransferFcn: '<S1>/Discrete Transfer Fcn' *)
           #rtb_Gain := #FOPD_Input - (#d_TmpSignalConversio[1] * #DiscreteTransferFcnv);
           #rtb_Divide := (#c_TmpSignalConversio[0] * #rtb_Gain) + (#c_TmpSignalConversio[1] * #DiscreteTransferFcnv);
           (* Delay: '<S1>/Delay' *)
           IF #Dead_Time < 1.0 THEN
               (* Outport: '<Root>/FOPD_Output' *)
               #FOPD_Output := #rtb_Divide;
           ELSE
               IF #Dead_Time > 800.0 THEN
                   #b_i := 800;
               ELSE
                   #b_i := TRUNC(#Dead_Time);
               END_IF;
               (* Outport: '<Root>/FOPD_Output' *)
               #FOPD_Output := #Delay_DSTATE[800 - #b_i];
           END_IF;
           (* End of Delay: '<S1>/Delay' *)

           (* Update for DiscreteTransferFcn: '<S1>/Discrete Transfer Fcn' *)
           #DiscreteTransferFcnv := #rtb_Gain;
           (* Update for Delay: '<S1>/Delay' *)
           FOR #b_i := 0 TO 798 DO
               #Delay_DSTATE[#b_i] := #Delay_DSTATE[#b_i + 1];
           END_FOR;
           #Delay_DSTATE[799] := #rtb_Divide;
           (* End of Update for Delay: '<S1>/Delay' *)
   END_CASE;
END_FUNCTION_BLOCK

FUNCTION_BLOCK "c_Smith_Predictor_MI"   // FB6, SCL
{ S7_Optimized_Access := 'TRUE' }
VERSION : 0.1
   VAR_INPUT
      ssMethodType : Int;
      Setpoint : Real;
      Process_Value : Real;
      Gain_System : Real;
      Time_Constant_System : Real;
      Dead_Time_System : DInt;
      Enable_Auto : Real;
      Hand_Value : Real;
      P_Controller : Real;
      I_Controller : Real;
      Start_Identification : Real;
      c_Time_Constant_Gain : Real;
      c_Time_Constant_Esti : Real;
      Enable_Adaption : Real;
      Sample_Time : Real;
   END_VAR
   VAR_OUTPUT
      Gain_NOT_Filtered : Real;
      Gain_Filtered : Real;
      Controller_Value : Real;
   END_VAR
   VAR
      UnitDelay_DSTATE : Real;
      c_Integrator_IC_LOAD : Int;
      Integrator_DSTATE : Real;
      c_Integrator_PrevRes : Int;
      In1 : Real;
      In1_b : Real;
      icLoad : Int;
      icLoad_i : Int;
      icLoad_p : Int;
      icLoad_b : Int;
      icLoad_ih : Int;
      icLoad_n : Int;
      Multiply : Real;
      In1_a : Real;
      In1_n : Real;
      UnitDelay_DSTATE_j : Real;
      c_arxEstimator_not_e : Bool;
      arxEstimator : "c_d_recursiveEstimat";
      DiscreteTransferFcnv : Real;
      b_DiscreteTransferFc : Real;
      c_System_Delay_Simul : Int := 3;
      delayTheta_Reset_ZCE : Int := 3;
      delayL_Reset_ZCE : Int := 3;
      delayPhi_Reset_ZCE : Int := 3;
      c_delayBufferU_Reset : Int := 3;
      c_delayBufferY_Reset : Int := 3;
      c_delayBufferRegress : Int := 3;
      Delay_Reset_ZCE : Int := 3;
      d_System_Delay_Simul : Int := 3;
      c_DiscreteTransferFc : Int := 3;
      d_DiscreteTransferFc : Int := 3;
      e_System_Delay_Simul : Array[0..799] of Real;
      f_System_Delay_Simul : Array[0..799] of Real;
      c_TmpSignalConversio : Array[0..1] of Real;
      d_TmpSignalConversio : Array[0..1] of Real;
      e_TmpSignalConversio : Array[0..1] of Real;
      f_TmpSignalConversio : Array[0..1] of Real;
      delayL_DSTATE : Array[0..8] of Real;
      delayTheta_DSTATE : Array[0..2] of Real;
      delayPhi_DSTATE : Array[0..3] of Real;
      c_InitialCovariancev : Array[0..8] of Real;
      i0_ZCFCN_d_RISING : "ZCFCN_d_RISING";
      i0_PT1_Tustin1 : "PT1_Tustin1";
      i1_PT1_Tustin1 : "PT1_Tustin1";
      phi : Array[0..2] of Real;
      fTr : Array[0..2] of Real;
      a1 : Real;
      sqrtA0overA1 : Real;
      sqrtA0timesA1 : Real;
      b_kk : DInt;
      rtb_UnitDelay : Real;
      rtb_theta : Array[0..2] of Real;
      rtb_AzSumofElements : Real;
      c_rtb_DiscreteTransf : Real;
      d_rtb_DiscreteTransf : Real;
      rtb_L : Array[0..8] of Real;
      rtb_phiMemory : Array[0..3] of Real;
      rtb_theta_tmp : Real;
   END_VAR
   // c_InitialCovariancev[0] := 3.162278;
   // c_InitialCovariancev[1] := 0.0;
   // c_InitialCovariancev[2] := 0.0;
   // c_InitialCovariancev[3] := 0.0;
   // c_InitialCovariancev[4] := 3.162278;
   // c_InitialCovariancev[5] := 0.0;
   // c_InitialCovariancev[6] := 0.0;
   // c_InitialCovariancev[7] := 0.0;
   // c_InitialCovariancev[8] := 3.162278;
BEGIN
   CASE #ssMethodType OF
       0:
           (* InitializeConditions for UnitDelay: '<S1>/Unit Delay' *)
           #UnitDelay_DSTATE := 0.0;
           (* SystemInitialize for Atomic SubSystem: '<S1>/System Identification' *)
           (* InitializeConditions for Delay: '<S3>/System_Delay_Simulation' *)
           FOR #b_kk := 0 TO 799 DO
               #e_System_Delay_Simul[#b_kk] := 0.0;
           END_FOR;
           (* End of InitializeConditions for Delay: '<S3>/System_Delay_Simulation' *)

           (* InitializeConditions for Delay: '<S110>/delayTheta' *)
           #icLoad := 1;
           (* InitializeConditions for Delay: '<S110>/delayL' *)
           #icLoad_i := 1;
           (* InitializeConditions for Delay: '<S110>/delayPhi' *)
           #icLoad_p := 1;
           (* InitializeConditions for Delay: '<S110>/delayBufferU' *)
           #icLoad_b := 1;
           (* InitializeConditions for Delay: '<S110>/delayBufferY' *)
           #icLoad_ih := 1;
           (* InitializeConditions for Delay: '<S130>/delayBufferRegressors' *)
           #icLoad_n := 1;
           (* SystemInitialize for Enabled SubSystem: '<S3>/Get_Current_delayed_Input_Offset' *)
           (* SystemInitialize for Outport: '<S106>/Hold when disabled' *)
           #In1 := 0.0;
           (* End of SystemInitialize for SubSystem: '<S3>/Get_Current_delayed_Input_Offset' *)
           (* End of SystemInitialize for SubSystem: '<S1>/System Identification' *)

           (* Constant: '<S3>/Constant2' *)
           #i0_PT1_Tustin1(ssMethodType := 0,
                           PT1_Input := #a1,
                           Gain_System := 1.0,
                           Time_Constant_System := #c_Time_Constant_Esti,
                           Reset := #Start_Identification);
           (* SystemInitialize for Atomic SubSystem: '<S1>/System Identification' *)
           (* SystemInitialize for Enabled SubSystem: '<S3>/Get_Current_Output_Offset' *)
           (* SystemInitialize for Outport: '<S105>/Hold when disabled' *)
           #In1_b := 0.0;
           (* End of SystemInitialize for SubSystem: '<S3>/Get_Current_Output_Offset' *)
           (* End of SystemInitialize for SubSystem: '<S1>/System Identification' *)

           (* Constant: '<S3>/Constant2' *)
           #i1_PT1_Tustin1(ssMethodType := 0,
                           PT1_Input := #a1,
                           Gain_System := 1.0,
                           Time_Constant_System := #c_Time_Constant_Esti,
                           Reset := #Start_Identification);
           (* SystemInitialize for Atomic SubSystem: '<S1>/System Identification' *)
           (* SystemInitialize for MATLAB Function: '<S130>/rarx' *)
           #c_arxEstimator_not_e := FALSE;
           (* SystemInitialize for Atomic SubSystem: '<S3>/PT1_Tustin' *)
           (* InitializeConditions for DiscreteTransferFcn: '<S107>/Discrete Transfer Fcn' *)
           #DiscreteTransferFcnv := 0.0;
           (* End of SystemInitialize for SubSystem: '<S3>/PT1_Tustin' *)
           (* End of SystemInitialize for SubSystem: '<S1>/System Identification' *)

           (* SystemInitialize for Atomic SubSystem: '<S1>/Adaptive SmithPredictor1' *)
           (* InitializeConditions for UnitDelay: '<S2>/Unit Delay' *)
           #UnitDelay_DSTATE_j := 0.0;
           (* InitializeConditions for DiscreteIntegrator: '<S62>/Integrator' *)
           #c_Integrator_IC_LOAD := 1;
           #c_Integrator_PrevRes := 2;
           (* End of SystemInitialize for SubSystem: '<S1>/Adaptive SmithPredictor1' *)
           (* SystemInitialize for Atomic SubSystem: '<S1>/Adaptive SmithPredictor1' *)
           (* InitializeConditions for Delay: '<S2>/System_Delay_Simulation' *)
           FOR #b_kk := 0 TO 799 DO
               #f_System_Delay_Simul[#b_kk] := 0.0;
           END_FOR;
           (* End of InitializeConditions for Delay: '<S2>/System_Delay_Simulation' *)

           (* SystemInitialize for Enabled SubSystem: '<S2>/Get_Current_Offset1' *)
           (* SystemInitialize for Outport: '<S5>/Hold when disabled' *)
           #In1_a := 0.0;
           (* End of SystemInitialize for SubSystem: '<S2>/Get_Current_Offset1' *)

           (* SystemInitialize for Enabled SubSystem: '<S2>/Get_Current_Offset' *)
           (* SystemInitialize for Outport: '<S4>/Hold when disabled' *)
           #In1_n := 0.0;
           (* End of SystemInitialize for SubSystem: '<S2>/Get_Current_Offset' *)

           (* SystemInitialize for Atomic SubSystem: '<S2>/PT1_Tustin' *)
           (* InitializeConditions for DiscreteTransferFcn: '<S7>/Discrete Transfer Fcn' *)
           #b_DiscreteTransferFc := 0.0;
           (* End of SystemInitialize for SubSystem: '<S2>/PT1_Tustin' *)
           (* End of SystemInitialize for SubSystem: '<S1>/Adaptive SmithPredictor1' *)
       1:
           (* UnitDelay: '<S1>/Unit Delay' *)
           #rtb_UnitDelay := #UnitDelay_DSTATE;
           (* Outputs for Atomic SubSystem: '<S1>/System Identification' *)
           (* Delay: '<S3>/System_Delay_Simulation' incorporates:
            *  Constant: '<S3>/Vorsicht wenn resettet wird muss erst dieser Totzeitspeicher  voll gelaufen sein bevor die Adaption starten darf  Sonst kommt heir immer 0 raus und die Identifikation kann nicht rechnen' *)
           #i0_ZCFCN_d_RISING(u0 := #c_System_Delay_Simul,
                              u1 := 0.0);
           #b_kk := #i0_ZCFCN_d_RISING.y0;
           #c_System_Delay_Simul := #i0_ZCFCN_d_RISING.y1;
           IF #b_kk <> 0 THEN
               FOR #b_kk := 0 TO 799 DO
                   #e_System_Delay_Simul[#b_kk] := 0.0;
               END_FOR;
           END_IF;
           IF #Dead_Time_System <= 0 THEN
               #d_rtb_DiscreteTransf := #rtb_UnitDelay;
           ELSE
               IF #Dead_Time_System > 800 THEN
                   #b_kk := 800;
               ELSE
                   #b_kk := #Dead_Time_System;
               END_IF;
               #d_rtb_DiscreteTransf := #e_System_Delay_Simul[800 - #b_kk];
           END_IF;
           (* End of Delay: '<S3>/System_Delay_Simulation' *)

           (* Outputs for Enabled SubSystem: '<S3>/Get_Current_delayed_Input_Offset' incorporates:
            *  EnablePort: '<S106>/Enable' *)
            (* Logic: '<S3>/NOT1' incorporates:
             *  Inport: '<S106>/In1' *)
           IF #Start_Identification = 0.0 THEN
               #In1 := #d_rtb_DiscreteTransf;
           END_IF;
           (* End of Logic: '<S3>/NOT1' *)
           (* End of Outputs for SubSystem: '<S3>/Get_Current_delayed_Input_Offset' *)

           (* MATLAB Function: '<S130>/rarx' incorporates:
            *  Constant: '<S3>/Constant2'
            *  Sum: '<S3>/Substract Current Offset  so that the linearised model works1' *)
           #i0_PT1_Tustin1(ssMethodType := 3,
                           PT1_Input := #d_rtb_DiscreteTransf - #In1,
                           Gain_System := 1.0,
                           Time_Constant_System := #c_Time_Constant_Esti,
                           Reset := #Start_Identification);
           #rtb_phiMemory[2] := #i0_PT1_Tustin1.PT1_Output;
           (* Outputs for Enabled SubSystem: '<S3>/Get_Current_Output_Offset' incorporates:
            *  EnablePort: '<S105>/Enable' *)
            (* Logic: '<S3>/NOT' incorporates:
             *  Inport: '<S105>/In1' *)
           IF #Start_Identification = 0.0 THEN
               #In1_b := #Process_Value;
           END_IF;
           (* End of Logic: '<S3>/NOT' *)
           (* End of Outputs for SubSystem: '<S3>/Get_Current_Output_Offset' *)

           (* Sum: '<S3>/Substract Current Offset  so that the linearised model works' incorporates:
            *  Constant: '<S3>/Constant2' *)
           #i1_PT1_Tustin1(ssMethodType := 3,
                           PT1_Input := #Process_Value - #In1_b,
                           Gain_System := 1.0,
                           Time_Constant_System := #c_Time_Constant_Esti,
                           Reset := #Start_Identification);
           #d_rtb_DiscreteTransf := #i1_PT1_Tustin1.PT1_Output;
           (* Delay: '<S110>/delayTheta' *)
           #i0_ZCFCN_d_RISING(u0 := #delayTheta_Reset_ZCE,
                              u1 := #Start_Identification);
           #b_kk := #i0_ZCFCN_d_RISING.y0;
           #delayTheta_Reset_ZCE := #i0_ZCFCN_d_RISING.y1;
           IF #b_kk <> 0 THEN
               #icLoad := 1;
           END_IF;
           IF #icLoad <> 0 THEN
               #delayTheta_DSTATE[0] := 2.2204460492503131E-16;
               #delayTheta_DSTATE[1] := 2.2204460492503131E-16;
               #delayTheta_DSTATE[2] := 2.2204460492503131E-16;
           END_IF;
           (* Delay: '<S110>/delayL' incorporates:
            *  Constant: '<S110>/InitialCovariance' *)
           #i0_ZCFCN_d_RISING(u0 := #delayL_Reset_ZCE,
                              u1 := #Start_Identification);
           #b_kk := #i0_ZCFCN_d_RISING.y0;
           #delayL_Reset_ZCE := #i0_ZCFCN_d_RISING.y1;
           IF #b_kk <> 0 THEN
               #icLoad_i := 1;
           END_IF;
           IF #icLoad_i <> 0 THEN
               FOR #b_kk := 0 TO 8 DO
                   #delayL_DSTATE[#b_kk] := #c_InitialCovariancev[#b_kk];
               END_FOR;
           END_IF;
           (* Delay: '<S110>/delayPhi' *)
           #i0_ZCFCN_d_RISING(u0 := #delayPhi_Reset_ZCE,
                              u1 := #Start_Identification);
           #b_kk := #i0_ZCFCN_d_RISING.y0;
           #delayPhi_Reset_ZCE := #i0_ZCFCN_d_RISING.y1;
           IF #b_kk <> 0 THEN
               #icLoad_p := 1;
           END_IF;
           IF #icLoad_p <> 0 THEN
               #delayPhi_DSTATE[0] := 0.0;
               #delayPhi_DSTATE[1] := 0.0;
               #delayPhi_DSTATE[2] := 0.0;
               #delayPhi_DSTATE[3] := 0.0;
           END_IF;
           (* Delay: '<S110>/delayBufferU' *)
           #i0_ZCFCN_d_RISING(u0 := #c_delayBufferU_Reset,
                              u1 := #Start_Identification);
           #b_kk := #i0_ZCFCN_d_RISING.y0;
           #c_delayBufferU_Reset := #i0_ZCFCN_d_RISING.y1;
           IF #b_kk <> 0 THEN
               #icLoad_b := 1;
           END_IF;
           (* End of Delay: '<S110>/delayBufferU' *)

           (* Delay: '<S110>/delayBufferY' *)
           #i0_ZCFCN_d_RISING(u0 := #c_delayBufferY_Reset,
                              u1 := #Start_Identification);
           #b_kk := #i0_ZCFCN_d_RISING.y0;
           #c_delayBufferY_Reset := #i0_ZCFCN_d_RISING.y1;
           IF #b_kk <> 0 THEN
               #icLoad_ih := 1;
           END_IF;
           (* End of Delay: '<S110>/delayBufferY' *)

           (* Delay: '<S130>/delayBufferRegressors' *)
           #i0_ZCFCN_d_RISING(u0 := #c_delayBufferRegress,
                              u1 := #Start_Identification);
           #b_kk := #i0_ZCFCN_d_RISING.y0;
           #c_delayBufferRegress := #i0_ZCFCN_d_RISING.y1;
           IF #b_kk <> 0 THEN
               #icLoad_n := 1;
           END_IF;
           (* End of Delay: '<S130>/delayBufferRegressors' *)

           (* Delay: '<S132>/Delay' *)
           #i0_ZCFCN_d_RISING(u0 := #Delay_Reset_ZCE,
                              u1 := #Start_Identification);
           #b_kk := #i0_ZCFCN_d_RISING.y0;
           #Delay_Reset_ZCE := #i0_ZCFCN_d_RISING.y1;
           (* MATLAB Function: '<S130>/rarx' *)
           (* % Was a reset trigered? *)
           (* MATLAB Function 'Recursive Estimation/rarx/rarx': '<S139>:1' *)
           (* Copyright 2015-2018 The MathWorks, Inc. *)
           (* Get the estimator object. Use the arx estimator with nb=0 *)
           (* '<S139>:1:17' if isempty(arxEstimator) *)
           IF NOT #c_arxEstimator_not_e THEN
               (* '<S139>:1:18' arxEstimator = recursiveEstimation.internal.rpoly.getEstimator(... *)
               (* '<S139>:1:19'         'arx',... *)
               (* '<S139>:1:20'         algorithmParams); *)
               #c_arxEstimator_not_e := TRUE;
           END_IF;
           (* If user triggered a reset, communicate this to the estimator *)
           (* '<S139>:1:24' if hasTriggeredReset *)
           (* Update algorithm states, perform estimation *)
           (* % States *)
           (* % new IO data *)
           (* '<S139>:1:31' [phiMemory, uMemory, yMemory, regressorsMemory, ... *)
           (* '<S139>:1:32'     theta, L, ... *)
           (* '<S139>:1:33'     A, B, e] = ... *)
           (* '<S139>:1:34'     arxEstimator.estimate(... *)
           (* '<S139>:1:35'     phiMemory, uMemory, yMemory, regressorsMemory, theta, L, ... % States *)
           (* '<S139>:1:36'     yMeas, uMeas,... % new IO data *)
           (* '<S139>:1:37'     isEnabled, adg1, adg2, algorithmParams); *)
           #arxEstimator.OutputDataIterator.IteratorPosition := 1;
           #arxEstimator.InputDataIterator.IteratorPosition := 1;
           #arxEstimator.OutputDataIterator.IteratorPosition := MIN(IN1 := #arxEstimator.OutputDataIterator.IteratorPosition + 1,
                                                                    IN2 := 2);
           #arxEstimator.InputDataIterator.IteratorPosition := MIN(IN1 := #arxEstimator.InputDataIterator.IteratorPosition + 1,
                                                                   IN2 := 2);
           (* End of Outputs for SubSystem: '<S1>/System Identification' *)
           (* Outputs for Atomic SubSystem: '<S1>/System Identification' *)
           (* MATLAB Function: '<S130>/rarx' incorporates:
            *  DataTypeConversion: '<S110>/DataTypeConversionEnable'
            *  Delay: '<S110>/delayL'
            *  Delay: '<S110>/delayPhi'
            *  Delay: '<S110>/delayTheta' *)
           FOR #b_kk := 0 TO 8 DO
               #rtb_L[#b_kk] := #delayL_DSTATE[#b_kk];
           END_FOR;
           #rtb_theta[0] := #delayTheta_DSTATE[0];
           #rtb_theta[1] := #delayTheta_DSTATE[1];
           #rtb_theta[2] := #delayTheta_DSTATE[2];
           #c_rtb_DiscreteTransf := #d_rtb_DiscreteTransf - (((#delayPhi_DSTATE[0] * #delayTheta_DSTATE[0]) + (#delayPhi_DSTATE[1] * #delayTheta_DSTATE[1])
           ) + (#delayPhi_DSTATE[3] * #delayTheta_DSTATE[2]));
           IF #Start_Identification <> 0.0 THEN
               FOR #b_kk := 0 TO 2 DO
                   #fTr[#b_kk] := (#delayL_DSTATE[(3 * #b_kk) + 2] * #delayPhi_DSTATE[3]) + ((#delayL_DSTATE[(3 * #b_kk) + 1] * #delayPhi_DSTATE[1])
                   + (#delayL_DSTATE[3 * #b_kk] * #delayPhi_DSTATE[0]));
               END_FOR;
               #phi[0] := 0.0;
               #rtb_theta[0] := 0.0;
               #phi[1] := 0.0;
               #rtb_theta[1] := 0.0;
               #a1 := (#fTr[2] * #fTr[2]) + 1.0;
               #sqrtA0overA1 := SQRT(1.0 / #a1);
               #rtb_theta[2] := #rtb_L[8] * #fTr[2];
               #rtb_L[8] := (#rtb_L[8] * #sqrtA0overA1) - (0.0 / (#sqrtA0overA1 * #a1));
               #phi[2] := #rtb_theta[2];
               #sqrtA0overA1 := #a1;
               #a1 := (#fTr[1] * #fTr[1]) + #a1;
               #sqrtA0overA1 := SQRT(#sqrtA0overA1 / #a1);
               #sqrtA0timesA1 := #sqrtA0overA1 * #a1;
               FOR #b_kk := 0 TO 1 DO
                   #rtb_AzSumofElements := #rtb_L[5 - #b_kk];
                   #rtb_theta_tmp := #phi[2 - #b_kk];
                   #rtb_theta[2 - #b_kk] := (#rtb_AzSumofElements * #fTr[1]) + #rtb_theta_tmp;
                   #rtb_L[5 - #b_kk] := (#rtb_AzSumofElements * #sqrtA0overA1) - ((#rtb_theta_tmp * #fTr[1]) / #sqrtA0timesA1);
                   #phi[2 - #b_kk] := #rtb_theta[2 - #b_kk];
               END_FOR;
               #sqrtA0overA1 := #a1;
               #a1 := (#fTr[0] * #fTr[0]) + #a1;
               #sqrtA0overA1 := SQRT(#sqrtA0overA1 / #a1);
               #sqrtA0timesA1 := #sqrtA0overA1 * #a1;
               FOR #b_kk := 0 TO 2 DO
                   #rtb_AzSumofElements := #rtb_L[2 - #b_kk];
                   #rtb_theta_tmp := #phi[2 - #b_kk];
                   #rtb_theta[2 - #b_kk] := (#rtb_AzSumofElements * #fTr[0]) + #rtb_theta_tmp;
                   #rtb_L[2 - #b_kk] := (#rtb_AzSumofElements * #sqrtA0overA1) - ((#rtb_theta_tmp * #fTr[0]) / #sqrtA0timesA1);
                   #phi[2 - #b_kk] := #rtb_theta[2 - #b_kk];
               END_FOR;
               #rtb_theta[0] := #rtb_theta[0] / #a1;
               #rtb_theta[1] := #rtb_theta[1] / #a1;
               #rtb_theta[0] := (#rtb_theta[0] * #c_rtb_DiscreteTransf) + #delayTheta_DSTATE[0];
               #rtb_theta[1] := (#rtb_theta[1] * #c_rtb_DiscreteTransf) + #delayTheta_DSTATE[1];
               #rtb_theta[2] := ((#rtb_theta[2] / #a1) * #c_rtb_DiscreteTransf) + #delayTheta_DSTATE[2];
           END_IF;
           #rtb_phiMemory[3] := #rtb_phiMemory[2];
           #rtb_phiMemory[2] := #delayPhi_DSTATE[1];
           #rtb_phiMemory[1] := #delayPhi_DSTATE[0];
           #rtb_phiMemory[0] := - #d_rtb_DiscreteTransf;
           (* Outputs for Atomic SubSystem: '<S3>/Calculate DC Gain1' *)
           (* Product: '<S104>/Divide' incorporates:
            *  MATLAB Function: '<S130>/rarx'
            *  Sum: '<S104>/A(z) Sum of Elements' *)
            (* helper variables *)
           #d_rtb_DiscreteTransf := #rtb_theta[2] / ((1.0 + #rtb_theta[0]) + #rtb_theta[1]);
           (* Saturate: '<S104>/Gain_Saturation' *)
           IF #d_rtb_DiscreteTransf >= 1.5 THEN
               #Gain_NOT_Filtered := 1.5;
           ELSIF #d_rtb_DiscreteTransf > 0.01 THEN
               #Gain_NOT_Filtered := #d_rtb_DiscreteTransf;
           ELSE
               #Gain_NOT_Filtered := 0.01;
           END_IF;
           (* End of Saturate: '<S104>/Gain_Saturation' *)
           (* End of Outputs for SubSystem: '<S3>/Calculate DC Gain1' *)

           (* Outputs for Atomic SubSystem: '<S3>/PT1_Tustin' *)
           (* Gain: '<S107>/Gain' *)
           #sqrtA0overA1 := 2.0 * #c_Time_Constant_Gain;
           (* Product: '<S107>/Multiply' incorporates:
            *  Constant: '<S3>/Constant' *)
           #Multiply := 1.0;
           (* Product: '<S107>/Divide' incorporates:
            *  Constant: '<S3>/Constant'
            *  Sum: '<S107>/Add' *)
           #d_rtb_DiscreteTransf := #Multiply / (1.0 + #sqrtA0overA1);
           (* SignalConversion: '<S107>/TmpSignal ConversionAtDiscrete Transfer FcnInport2' *)
           #c_TmpSignalConversio[0] := #d_rtb_DiscreteTransf;
           #c_TmpSignalConversio[1] := #d_rtb_DiscreteTransf;
           (* SignalConversion: '<S107>/TmpSignal ConversionAtDiscrete Transfer FcnInport3' incorporates:
            *  Constant: '<S107>/Constant'
            *  Constant: '<S3>/Constant'
            *  Gain: '<S107>/Gain1'
            *  Product: '<S107>/Divide1'
            *  Sum: '<S107>/Add1'
            *  Sum: '<S107>/Minus' *)
           #d_TmpSignalConversio[0] := 1.0;
           #d_TmpSignalConversio[1] := - ((#sqrtA0overA1 - 1.0) / (#sqrtA0overA1 + 1.0));
           (* DiscreteTransferFcn: '<S107>/Discrete Transfer Fcn' *)
           #i0_ZCFCN_d_RISING(u0 := #c_DiscreteTransferFc,
                              u1 := #Start_Identification);
           #b_kk := #i0_ZCFCN_d_RISING.y0;
           #c_DiscreteTransferFc := #i0_ZCFCN_d_RISING.y1;
           IF #b_kk <> 0 THEN
               #DiscreteTransferFcnv := 0.0;
           END_IF;
           #d_rtb_DiscreteTransf := #Gain_NOT_Filtered - (#d_TmpSignalConversio[1] * #DiscreteTransferFcnv);
           #sqrtA0timesA1 := (#c_TmpSignalConversio[0] * #d_rtb_DiscreteTransf) + (#c_TmpSignalConversio[1] * #DiscreteTransferFcnv)
           ;
           (* End of DiscreteTransferFcn: '<S107>/Discrete Transfer Fcn' *)

           (* Update for DiscreteTransferFcn: '<S107>/Discrete Transfer Fcn' *)
           #DiscreteTransferFcnv := #d_rtb_DiscreteTransf;
           (* End of Outputs for SubSystem: '<S3>/PT1_Tustin' *)

           (* Update for Delay: '<S3>/System_Delay_Simulation' *)
           FOR #b_kk := 0 TO 798 DO
               #e_System_Delay_Simul[#b_kk] := #e_System_Delay_Simul[#b_kk + 1];
           END_FOR;
           #e_System_Delay_Simul[799] := #rtb_UnitDelay;
           (* End of Update for Delay: '<S3>/System_Delay_Simulation' *)

           (* Update for Delay: '<S110>/delayTheta' *)
           #icLoad := 0;
           #delayTheta_DSTATE[0] := #rtb_theta[0];
           #delayTheta_DSTATE[1] := #rtb_theta[1];
           #delayTheta_DSTATE[2] := #rtb_theta[2];
           (* Update for Delay: '<S110>/delayL' *)
           #icLoad_i := 0;
           (* End of Outputs for SubSystem: '<S1>/System Identification' *)
           (* Outputs for Atomic SubSystem: '<S1>/System Identification' *)
           (* Update for Delay: '<S110>/delayL' *)
           FOR #b_kk := 0 TO 8 DO
               #delayL_DSTATE[#b_kk] := #rtb_L[#b_kk];
           END_FOR;
           (* Update for Delay: '<S110>/delayPhi' *)
           #icLoad_p := 0;
           #delayPhi_DSTATE[0] := #rtb_phiMemory[0];
           #delayPhi_DSTATE[1] := #rtb_phiMemory[1];
           #delayPhi_DSTATE[2] := #rtb_phiMemory[2];
           #delayPhi_DSTATE[3] := #rtb_phiMemory[3];
           (* Update for Delay: '<S110>/delayBufferU' *)
           #icLoad_b := 0;
           (* Update for Delay: '<S110>/delayBufferY' *)
           #icLoad_ih := 0;
           (* Update for Delay: '<S130>/delayBufferRegressors' *)
           #icLoad_n := 0;
           (* End of Outputs for SubSystem: '<S1>/System Identification' *)

           (* Outport: '<Root>/Gain_Filtered' *)
           #Gain_Filtered := #sqrtA0timesA1;
           (* Outputs for Atomic SubSystem: '<S1>/Adaptive SmithPredictor1' *)
           (* Switch: '<S2>/Check if Controller  Integrator is 0' incorporates:
            *  Constant: '<S2>/Constant'
            *  Constant: '<S2>/Constant6'
            *  Product: '<S2>/Invert Integrator' *)
           IF #I_Controller <> 0.0 THEN
               #d_rtb_DiscreteTransf := 1.0 / #I_Controller;
           ELSE
               #d_rtb_DiscreteTransf := 0.0;
           END_IF;
           (* End of Switch: '<S2>/Check if Controller  Integrator is 0' *)

           (* Product: '<S2>/Divide' *)
           #rtb_AzSumofElements := #Hand_Value / #P_Controller;
           (* Switch: '<S2>/Hand_Mode2' incorporates:
            *  Constant: '<S2>/Constant2' *)
           IF #Enable_Auto > 0.0 THEN
               #sqrtA0overA1 := #Setpoint;
           ELSE
               #sqrtA0overA1 := 0.0;
           END_IF;
           (* End of Switch: '<S2>/Hand_Mode2' *)

           (* Outputs for Enabled SubSystem: '<S2>/Get_Current_Offset1' incorporates:
            *  EnablePort: '<S5>/Enable' *)
            (* Logic: '<S2>/NOT1' incorporates:
             *  Inport: '<S5>/In1' *)
           IF #Enable_Auto = 0.0 THEN
               #In1_a := #Process_Value;
           END_IF;
           (* End of Logic: '<S2>/NOT1' *)
           (* End of Outputs for SubSystem: '<S2>/Get_Current_Offset1' *)

           (* Switch: '<S2>/Hand_Mode4' incorporates:
            *  Constant: '<S2>/Constant5' *)
           IF #Enable_Auto > 0.0 THEN
               #rtb_UnitDelay := #In1_a;
           ELSE
               #rtb_UnitDelay := 0.0;
           END_IF;
           (* End of Switch: '<S2>/Hand_Mode4' *)

           (* Sum: '<S2>/Sum' incorporates:
            *  Sum: '<S2>/Substract Current Setpoint Offset'
            *  UnitDelay: '<S2>/Unit Delay' *)
           #sqrtA0overA1 := (#sqrtA0overA1 - #rtb_UnitDelay) - #UnitDelay_DSTATE_j;
           (* DiscreteIntegrator: '<S62>/Integrator' *)
           IF #c_Integrator_IC_LOAD <> 0 THEN
               #Integrator_DSTATE := #rtb_AzSumofElements;
           END_IF;
           IF (#Enable_Auto > 0.0) AND (#c_Integrator_PrevRes <= 0) THEN
               #Integrator_DSTATE := #rtb_AzSumofElements;
           END_IF;
           (* Product: '<S53>/PProd Out' incorporates:
            *  DiscreteIntegrator: '<S62>/Integrator'
            *  Sum: '<S91>/Sum' *)
           #a1 := (#sqrtA0overA1 + #Integrator_DSTATE) * #P_Controller;
           (* Saturate: '<S83>/Saturation' *)
           IF #a1 >= 100.0 THEN
               #a1 := 100.0;
           ELSIF #a1 <= 0.0 THEN
               #a1 := 0.0;
           END_IF;
           (* End of Saturate: '<S83>/Saturation' *)

           (* Switch: '<S2>/Hand_Mode' *)
           IF #Enable_Auto > 0.0 THEN
               #Controller_Value := #a1;
           ELSE
               #Controller_Value := #Hand_Value;
           END_IF;
           (* End of Switch: '<S2>/Hand_Mode' *)

           (* Outputs for Enabled SubSystem: '<S2>/Get_Current_Offset' incorporates:
            *  EnablePort: '<S4>/Enable' *)
            (* Logic: '<S2>/NOT' incorporates:
             *  Inport: '<S4>/In1' *)
           IF #Enable_Auto = 0.0 THEN
               #In1_n := #Controller_Value;
           END_IF;
           (* End of Logic: '<S2>/NOT' *)
           (* End of Outputs for SubSystem: '<S2>/Get_Current_Offset' *)

           (* Switch: '<S2>/Hand_Mode1' incorporates:
            *  Constant: '<S2>/Constant3'
            *  Constant: '<S2>/Constant4'
            *  Sum: '<S2>/Substract Current Offset  so that the linearised model works'
            *  Switch: '<S2>/Hand_Mode3' *)
           IF #Enable_Auto > 0.0 THEN
               #a1 := #Controller_Value - #In1_n;
               #rtb_AzSumofElements := #Process_Value;
           ELSE
               #a1 := 0.0;
               #rtb_AzSumofElements := 0.0;
           END_IF;
           (* End of Switch: '<S2>/Hand_Mode1' *)

           (* Switch: '<S2>/Switch_from_initial_Gain_to_Estimated' *)
           IF #Enable_Adaption <= 0.0 THEN
               #sqrtA0timesA1 := #Gain_System;
           END_IF;
           (* End of Switch: '<S2>/Switch_from_initial_Gain_to_Estimated' *)

           (* Product: '<S2>/Mul_Gain_or_Estimate' *)
           #c_rtb_DiscreteTransf := #a1 * #sqrtA0timesA1;
           (* Outputs for Atomic SubSystem: '<S2>/PT1_Tustin' *)
           (* Gain: '<S7>/Gain' *)
           #sqrtA0timesA1 := 2.0 * #Time_Constant_System;
           (* Product: '<S7>/Divide' incorporates:
            *  Product: '<S7>/Multiply'
            *  Sum: '<S7>/Add' *)
           #a1 := #Sample_Time / (#Sample_Time + #sqrtA0timesA1);
           (* SignalConversion: '<S7>/TmpSignal ConversionAtDiscrete Transfer FcnInport2' *)
           #e_TmpSignalConversio[0] := #a1;
           #e_TmpSignalConversio[1] := #a1;
           (* SignalConversion: '<S7>/TmpSignal ConversionAtDiscrete Transfer FcnInport3' incorporates:
            *  Constant: '<S7>/Constant'
            *  Gain: '<S7>/Gain1'
            *  Product: '<S7>/Divide1'
            *  Sum: '<S7>/Add1'
            *  Sum: '<S7>/Minus' *)
           #f_TmpSignalConversio[0] := 1.0;
           #f_TmpSignalConversio[1] := - ((#sqrtA0timesA1 - #Sample_Time) / (#sqrtA0timesA1 + #Sample_Time));
           (* DiscreteTransferFcn: '<S7>/Discrete Transfer Fcn' *)
           #i0_ZCFCN_d_RISING(u0 := #d_DiscreteTransferFc,
                              u1 := #Enable_Auto);
           #b_kk := #i0_ZCFCN_d_RISING.y0;
           #d_DiscreteTransferFc := #i0_ZCFCN_d_RISING.y1;
           IF #b_kk <> 0 THEN
               #b_DiscreteTransferFc := 0.0;
           END_IF;
           #sqrtA0timesA1 := #c_rtb_DiscreteTransf - (#f_TmpSignalConversio[1] * #b_DiscreteTransferFc);
           #a1 := (#e_TmpSignalConversio[0] * #sqrtA0timesA1) + (#e_TmpSignalConversio[1] * #b_DiscreteTransferFc);
           (* End of DiscreteTransferFcn: '<S7>/Discrete Transfer Fcn' *)

           (* Update for DiscreteTransferFcn: '<S7>/Discrete Transfer Fcn' *)
           #b_DiscreteTransferFc := #sqrtA0timesA1;
           (* End of Outputs for SubSystem: '<S2>/PT1_Tustin' *)

           (* Delay: '<S2>/System_Delay_Simulation' *)
           #i0_ZCFCN_d_RISING(u0 := #d_System_Delay_Simul,
                              u1 := #Enable_Auto);
           #b_kk := #i0_ZCFCN_d_RISING.y0;
           #d_System_Delay_Simul := #i0_ZCFCN_d_RISING.y1;
           IF #b_kk <> 0 THEN
               FOR #b_kk := 0 TO 799 DO
                   #f_System_Delay_Simul[#b_kk] := 0.0;
               END_FOR;
           END_IF;
           IF #Dead_Time_System <= 0 THEN
               #sqrtA0timesA1 := #a1;
           ELSE
               IF #Dead_Time_System > 800 THEN
                   #b_kk := 800;
               ELSE
                   #b_kk := #Dead_Time_System;
               END_IF;
               #sqrtA0timesA1 := #f_System_Delay_Simul[800 - #b_kk];
           END_IF;
           (* End of Delay: '<S2>/System_Delay_Simulation' *)

           (* Update for UnitDelay: '<S2>/Unit Delay' incorporates:
            *  Sum: '<S2>/Substract Current Offset  so that the linearised model works1'
            *  Sum: '<S2>/Sum17'
            *  Sum: '<S2>/Sum18' *)
           #UnitDelay_DSTATE_j := ((#rtb_AzSumofElements - #rtb_UnitDelay) - #sqrtA0timesA1) + #a1;
           (* Update for DiscreteIntegrator: '<S62>/Integrator' incorporates:
            *  Product: '<S51>/IProd Out' *)
           #c_Integrator_IC_LOAD := 0;
           #Integrator_DSTATE := (#sqrtA0overA1 * #d_rtb_DiscreteTransf) + #Integrator_DSTATE;
           IF #Enable_Auto > 0.0 THEN
               #c_Integrator_PrevRes := 1;
           ELSIF #Enable_Auto < 0.0 THEN
               #c_Integrator_PrevRes := -1;
           ELSIF #Enable_Auto = 0.0 THEN
               #c_Integrator_PrevRes := 0;
           ELSE
               #c_Integrator_PrevRes := 2;
           END_IF;
           (* End of Update for DiscreteIntegrator: '<S62>/Integrator' *)

           (* Update for Delay: '<S2>/System_Delay_Simulation' *)
           FOR #b_kk := 0 TO 798 DO
               #f_System_Delay_Simul[#b_kk] := #f_System_Delay_Simul[#b_kk + 1];
           END_FOR;
           #f_System_Delay_Simul[799] := #a1;
           (* End of Update for Delay: '<S2>/System_Delay_Simulation' *)
           (* End of Outputs for SubSystem: '<S1>/Adaptive SmithPredictor1' *)

           (* Update for UnitDelay: '<S1>/Unit Delay' *)
           #UnitDelay_DSTATE := #Controller_Value;
   END_CASE;
END_FUNCTION_BLOCK

FUNCTION_BLOCK "b_ZCFCN_d_RISING"   // FB7, SCL
{ S7_Optimized_Access := 'TRUE' }
VERSION : 0.1
   VAR_INPUT
      u0 : Int;
      u1 : Real;
   END_VAR
   VAR_OUTPUT
      y0 : DInt;
      y1 : Int;
   END_VAR
   VAR
      rising : Bool;
      temp1 : Bool;
      temp2 : Bool;
   END_VAR
BEGIN
   #temp1 := FALSE;
   IF #u1 > 0.0 THEN
       #y1 := 1;
   ELSIF #u1 < 0.0 THEN
       #y1 := 2;
   ELSE
       #y1 := 0;
   END_IF;
   #temp2 := FALSE;
   IF #u0 = 2 THEN
       IF #y1 = 0 THEN
           #rising := TRUE;
       ELSIF #y1 = 1 THEN
           #rising := TRUE;
       ELSE
           #temp2 := TRUE;
       END_IF;
   ELSE
       #temp2 := TRUE;
   END_IF;
   IF #temp2 THEN
       IF #u0 = 0 THEN
           IF #y1 = 1 THEN
               #rising := TRUE;
           ELSE
               #temp1 := TRUE;
           END_IF;
       ELSE
           #temp1 := TRUE;
       END_IF;
   END_IF;
   IF #temp1 THEN
       IF #u0 = 101 THEN
           IF #y1 = 1 THEN
               #rising := TRUE;
           ELSE
               #rising := FALSE;
           END_IF;
       ELSE
           #rising := FALSE;
       END_IF;
   END_IF;
   IF #rising THEN
       #y0 := 1;
   ELSE
       #y0 := 0;
   END_IF;
   IF (#u0 = 2) AND (#y1 = 0) THEN
       #y1 := 100;
   END_IF;
END_FUNCTION_BLOCK

FUNCTION_BLOCK "PT1_Tustin1"   // FB8, SCL
{ S7_Optimized_Access := 'TRUE' }
VERSION : 0.1
   VAR_INPUT
      ssMethodType : Int;
      PT1_Input : Real;
      Gain_System : Real;
      Time_Constant_System : Real;
      Reset : Real;
   END_VAR
   VAR_OUTPUT
      PT1_Output : Real;
   END_VAR
   VAR
      Multiply : Real;
      DiscreteTransferFcnv : Real;
      b_DiscreteTransferFc : Int := 3;
      c_TmpSignalConversio : Array[0..1] of Real;
      d_TmpSignalConversio : Array[0..1] of Real;
      i0_b_ZCFCN_d_RISING : "b_ZCFCN_d_RISING";
      tempOutEvent : DInt;
      rtb_Gain_l : Real;
      rtb_Divide_p : Real;
   END_VAR
BEGIN
   CASE #ssMethodType OF
       0:
           (* InitializeConditions for DiscreteTransferFcn: '<S108>/Discrete Transfer Fcn' *)
           #DiscreteTransferFcnv := 0.0;
       3:
           (* Gain: '<S108>/Gain' *)
           #rtb_Gain_l := 2.0 * #Time_Constant_System;
           (* Product: '<S108>/Multiply' *)
           #Multiply := #Gain_System * #Gain_System;
           (* Product: '<S108>/Divide' incorporates:
            *  Sum: '<S108>/Add' *)
           #rtb_Divide_p := #Multiply / (#Gain_System + #rtb_Gain_l);
           (* SignalConversion: '<S108>/TmpSignal ConversionAtDiscrete Transfer FcnInport2' *)
           #c_TmpSignalConversio[0] := #rtb_Divide_p;
           #c_TmpSignalConversio[1] := #rtb_Divide_p;
           (* SignalConversion: '<S108>/TmpSignal ConversionAtDiscrete Transfer FcnInport3' incorporates:
            *  Constant: '<S108>/Constant'
            *  Gain: '<S108>/Gain1'
            *  Product: '<S108>/Divide1'
            *  Sum: '<S108>/Add1'
            *  Sum: '<S108>/Minus' *)
           #d_TmpSignalConversio[0] := 1.0;
           #d_TmpSignalConversio[1] := - ((#rtb_Gain_l - #Gain_System) / (#rtb_Gain_l + #Gain_System));
           (* DiscreteTransferFcn: '<S108>/Discrete Transfer Fcn' *)
           #i0_b_ZCFCN_d_RISING(u0 := #b_DiscreteTransferFc,
                                u1 := #Reset);
           #tempOutEvent := #i0_b_ZCFCN_d_RISING.y0;
           #b_DiscreteTransferFc := #i0_b_ZCFCN_d_RISING.y1;
           IF #tempOutEvent <> 0 THEN
               #DiscreteTransferFcnv := 0.0;
           END_IF;
           #rtb_Gain_l := #PT1_Input - (#d_TmpSignalConversio[1] * #DiscreteTransferFcnv);
           #PT1_Output := (#c_TmpSignalConversio[0] * #rtb_Gain_l) + (#c_TmpSignalConversio[1] * #DiscreteTransferFcnv);
           (* End of DiscreteTransferFcn: '<S108>/Discrete Transfer Fcn' *)

           (* Update for DiscreteTransferFcn: '<S108>/Discrete Transfer Fcn' *)
           #DiscreteTransferFcnv := #rtb_Gain_l;
   END_CASE;
END_FUNCTION_BLOCK

ORGANIZATION_BLOCK "Main"   // OB1, LAD, ProgramCycle
TITLE = "Main Program Sweep (Cycle)"
{ S7_Optimized_Access := 'TRUE' }
VERSION : 0.1
   VAR_INPUT
      Initial_Call : Bool;   // Initial call of this OB
      Remanence : Bool;   // =True, if remanent data are available
   END_VAR
BEGIN
END_ORGANIZATION_BLOCK

ORGANIZATION_BLOCK "Cyclic interrupt_100ms"   // OB30, FBD, CyclicInterrupt
{ S7_Optimized_Access := 'TRUE' }
VERSION : 0.1
   VAR_INPUT
      Initial_Call : Bool;   // Initial call of this OB
      Event_Count : Int;   // Events discarded
   END_VAR
BEGIN

REGION Network 1: PT1
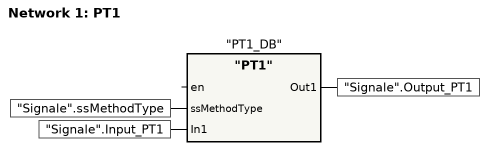
   "PT1_DB"(ssMethodType := "Signale".ssMethodType, In1 := "Signale".Input_PT1, Out1 => "Signale".Output_PT1);   // "PT1"
END_REGION

REGION Network 2: FOPDT
END_REGION
END_ORGANIZATION_BLOCK

ORGANIZATION_BLOCK "Cyclic interrupt_1s"   // OB31, FBD, CyclicInterrupt
{ S7_Optimized_Access := 'TRUE' }
VERSION : 0.1
   VAR_INPUT
      Initial_Call : Bool;   // Initial call of this OB
      Event_Count : Int;   // Events discarded
   END_VAR
BEGIN

REGION Network 1: Smith Predictor and Adaptive Gain
END_REGION

REGION Network 2
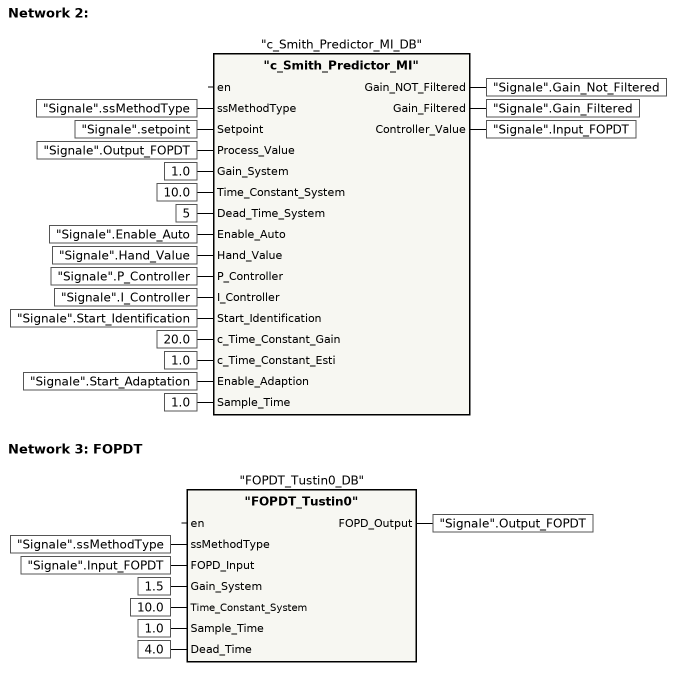
   "c_Smith_Predictor_MI_DB"(ssMethodType := "Signale".ssMethodType,   // "c_Smith_Predictor_MI"
                           Setpoint := "Signale".setpoint,
                           Process_Value := "Signale".Output_FOPDT,
                           Gain_System := 1.0,
                           Time_Constant_System := 10.0,
                           Dead_Time_System := 5,
                           Enable_Auto := "Signale".Enable_Auto,
                           Hand_Value := "Signale".Hand_Value,
                           P_Controller := "Signale".P_Controller,
                           I_Controller := "Signale".I_Controller,
                           Start_Identification := "Signale".Start_Identification,
                           c_Time_Constant_Gain := 20.0,
                           c_Time_Constant_Esti := 1.0,
                           Enable_Adaption := "Signale".Start_Adaptation,
                           Sample_Time := 1.0,
                           Gain_NOT_Filtered => "Signale".Gain_Not_Filtered,
                           Gain_Filtered => "Signale".Gain_Filtered,
                           Controller_Value => "Signale".Input_FOPDT);
END_REGION

REGION Network 3: FOPDT
   "FOPDT_Tustin0_DB"(ssMethodType := "Signale".ssMethodType,   // "FOPDT_Tustin0"
                      FOPD_Input := "Signale".Input_FOPDT,
                      Gain_System := 1.5,
                      Time_Constant_System := 10.0,
                      Sample_Time := 1.0,
                      Dead_Time := 4.0,
                      FOPD_Output => "Signale".Output_FOPDT);
END_REGION

REGION Network 4 (SCL): Pulse Indicator
   "Signale".pulse_Indicatior:= NOT "Signale".pulse_Indicatior;
END_REGION
END_ORGANIZATION_BLOCK